SUBAPPLICATION RedWhiteBackground2_AXC (* Hintergrundfarbe (TRUE -> Rot, FALSE -> Weiß) für 2 Objekte (AX-Adapter) (Kompakt) *)
  (* Standard: 61499-2 *)
  (* Version 1.0, 2026-07-21, franz, Meisterschulen am Ostbahnhof *)
  PACKAGE MyLib::sys;
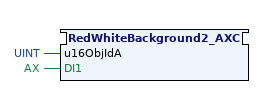
  VAR_INPUT
    u16ObjIdA : UINT;
  END_VAR
  SOCKETS
    DI1 : adapter::types::unidirectional::AX;
  END_SOCKETS
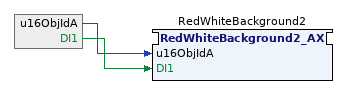
  SUBAPPS
    RedWhiteBackground2 : MyLib::sys::RedWhiteBackground2_AX;
  END_SUBAPPS
  DATA_CONNECTIONS
    u16ObjIdA TO RedWhiteBackground2.u16ObjIdA;
  END_CONNECTIONS
  ADAPTER_CONNECTIONS
    DI1 TO RedWhiteBackground2.DI1;
  END_CONNECTIONS
END_SUBAPPLICATION
